// TIA Portal V18 export
// export: Created 2026-06-09T02:47:53.128383Z, ExportSetting WithDefaults, DisplayName Totally Integrated Automation Portal, DisplayVersion V18, DisplayName TIA Portal Openness, DisplayVersion V18, DisplayName TIA Portal Version Control Interface, DisplayVersion V18, DisplayName STEP 7 Professional, DisplayVersion V18, DisplayName STEP 7 Safety, DisplayVersion V18, DisplayName WinCC Professional, DisplayVersion V18
FUNCTION_BLOCK "Pakowanie"   // FB4, LAD
{ S7_Optimized_Access := 'TRUE' }
VERSION : 0.1
// stored: AutoNumber true, IsIECCheckEnabled false, IsRetainMemResEnabled false, MemoryReserve 100, SetENOAutomatically false, UDAEnableTagReadback false
BEGIN

REGION Network 1
   // Start przenośnika taśmowego i zapalenie się lampy sygnalizacyjnej.
   // Wyłącznik pakowania znajduje się fizycznie na linii produkcyjnej, w jego skład wchodzi również kurtyna świetlna. Stop natomiast w panelu HMI.
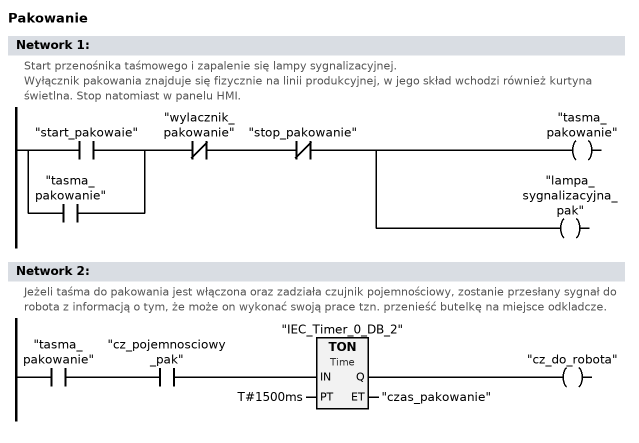
   RUNG wire#powerrail
      Contact( "start_pakowaie" )
      wire#w1
      I_Contact( "wylacznik_pakowanie" )
      I_Contact( "stop_pakowanie" )
      wire#w2
      Coil( "tasma_pakowanie" )
   END_RUNG
   RUNG wire#powerrail
      Contact( "tasma_pakowanie" )
   END_RUNG wire#w1
   RUNG wire#w2
      Coil( "lampa_sygnalizacyjna_pak" )
   END_RUNG
   // the same network as SCL:
   "tasma_pakowanie" := ("start_pakowaie" OR "tasma_pakowanie") AND NOT "wylacznik_pakowanie" AND NOT "stop_pakowanie";
   "lampa_sygnalizacyjna_pak" := "tasma_pakowanie";
END_REGION

REGION Network 2
   // Jeżeli taśma do pakowania jest włączona oraz zadziała czujnik pojemnościowy, zostanie przesłany sygnał do robota z informacją o tym, że może on wykonać swoją prace tzn. przenieść butelkę na miejsce odkladcze.
   RUNG wire#powerrail
      Contact( "tasma_pakowanie" )
      Contact( "cz_pojemnosciowy_pak" )
      { S7_Templates := "time_type := Time" } "IEC_Timer_0_DB_2".TON(pt := T#1500ms, et => "czas_pakowanie")
      Coil( "cz_do_robota" )
   END_RUNG
   // the same network as SCL:
   "IEC_Timer_0_DB_2".TON(IN := "tasma_pakowanie" AND "cz_pojemnosciowy_pak",
                          PT := T#1500ms,
                          ET => "czas_pakowanie");
   "cz_do_robota" := "IEC_Timer_0_DB_2".Q;
END_REGION
END_FUNCTION_BLOCK
